// TIA Portal V19 export
DATA_BLOCK "Alarms"   // DB88
// stored: MemoryReserve 100, Namespace Unit3.EM1
   VAR
      emAlarms { ExternalWritable := 'False'} : Array[0.._.Unit3_NO_OF_EMs] of "LAF_typeAlarms";
      errorNoReaction { ExternalWritable := 'False'} : Array[0..9] of Bool;   // Error without further impact
      errorAbort { ExternalWritable := 'False'} : Array[0..9] of Bool;   // Error which aborts the whole Unit
      errorStop { ExternalWritable := 'False'} : Array[0..9] of Bool;   // Error which stops the whole Unit
      warningNoReaction { ExternalWritable := 'False'} : Array[0..9] of Bool;   // Warning which could lead to a error
      warningHold { ExternalWritable := 'False'} : Array[0..9] of Bool;   // Warning which holds the whole Unit
      warningSuspend { ExternalWritable := 'False'} : Array[0..9] of Bool;   // Warning which suspends the whole Unit
      information { ExternalWritable := 'False'} : Array[0..9] of Bool;   // Informations of the EM
      criteriaAnalysis { ExternalWritable := 'False'} : Array[0..9] of Bool;   // CriteriaAnalysis of the EM
   END_VAR
BEGIN
   information[0] := false;
END_DATA_BLOCK
